FUNCTION_BLOCK Enable_Motor
VAR_INPUT
END_VAR
VAR_OUTPUT
END_VAR
VAR
END_VAR

// NETWORK 1

END_FUNCTION_BLOCK

(* stored: Version 1.1.0.1, ProductVersion 3.1.4024.12
   POU Enable_Motor: Id {587b4295-7407-45b7-a824-5552096de12b}, SpecialFunc None *)
